Omron CX-Programmer project Китайский_паллетайзер_с_комментариями (CX-Programmer 9.41)

# PLC НовыйПЛК1: CP1E N60

## Global symbols (name address type ; comment)
0.00 BOOL  ; Переключатель Р-А Магазин поддонов
0.01 BOOL  ; КН Магазин поддонов ВНИЗ
0.02 BOOL  ; Маг ВВЕРХ
0.03 BOOL  ; Лапы ОТКР

## Program РВіМРт1 (cyclic task 0)

### Section Сегмент1

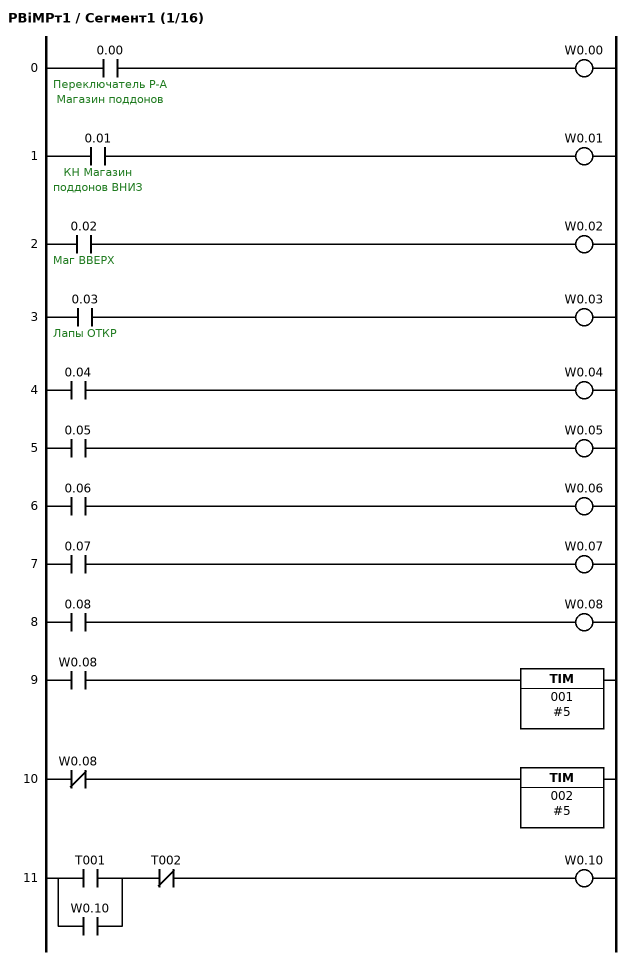
; rung 0
LD 0.00  ; Переключатель Р-А Магазин поддонов
OUT W0.00
; rung 1
LD 0.01  ; КН Магазин поддонов ВНИЗ
OUT W0.01
; rung 2
LD 0.02  ; Маг ВВЕРХ
OUT W0.02
; rung 3
LD 0.03  ; Лапы ОТКР
OUT W0.03
; rung 4
LD 0.04
OUT W0.04
; rung 5
LD 0.05
OUT W0.05
; rung 6
LD 0.06
OUT W0.06
; rung 7
LD 0.07
OUT W0.07
; rung 8
LD 0.08
OUT W0.08
; rung 9
LD W0.08
TIM 001 #5
; rung 10
LDNOT W0.08
TIM 002 #5
; rung 11
LD T001
OR W0.10
ANDNOT T002
OUT W0.10

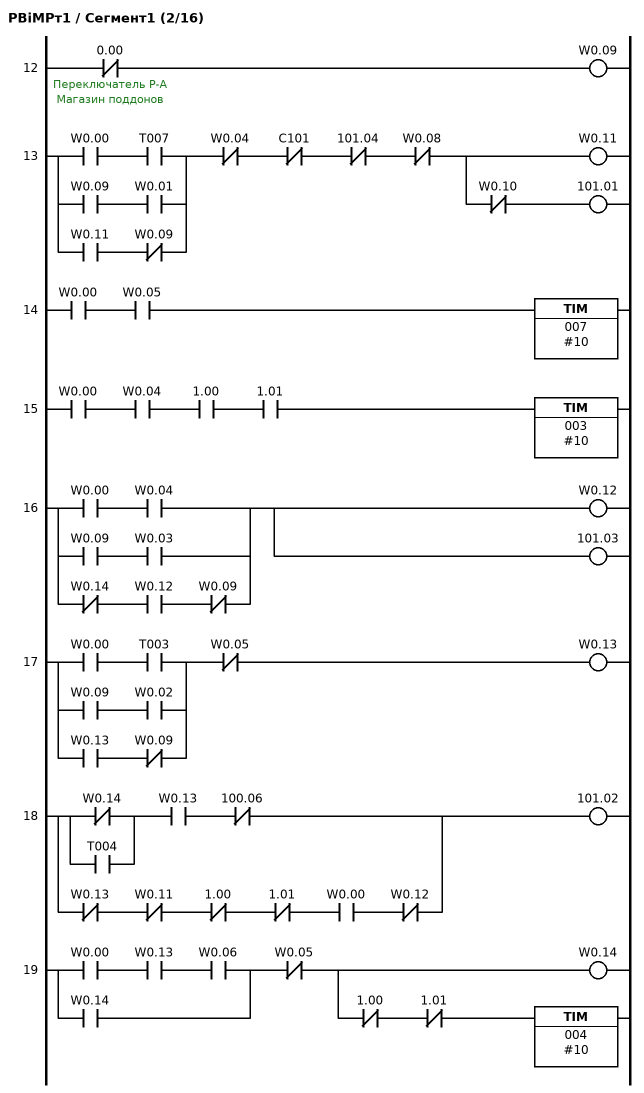
; rung 12
LDNOT 0.00  ; Переключатель Р-А Магазин поддонов
OUT W0.09
; rung 13
LD W0.00
AND T007
LD W0.09
AND W0.01
ORLD
LD W0.11
ANDNOT W0.09
ORLD
ANDNOT W0.04
ANDNOT C101
ANDNOT 101.04
ANDNOT W0.08
OUT W0.11
ANDNOT W0.10
OUT 101.01
; rung 14
LD W0.00
AND W0.05
TIM 007 #10
; rung 15
LD W0.00
AND W0.04
AND 1.00
AND 1.01
TIM 003 #10
; rung 16
LD W0.00
AND W0.04
LD W0.09
AND W0.03
ORLD
LDNOT W0.14
AND W0.12
ANDNOT W0.09
ORLD
OUT W0.12
OUT 101.03
; rung 17
LD W0.00
AND T003
LD W0.09
AND W0.02
ORLD
LD W0.13
ANDNOT W0.09
ORLD
ANDNOT W0.05
OUT W0.13
; rung 18
LDNOT W0.14
OR T004
AND W0.13
ANDNOT 100.06
LDNOT W0.13
ANDNOT W0.11
ANDNOT 1.00
ANDNOT 1.01
AND W0.00
ANDNOT W0.12
ORLD
OUT 101.02
; rung 19
LD W0.00
AND W0.13
AND W0.06
OR W0.14
ANDNOT W0.05
OUT W0.14
ANDNOT 1.00
ANDNOT 1.01
TIM 004 #10

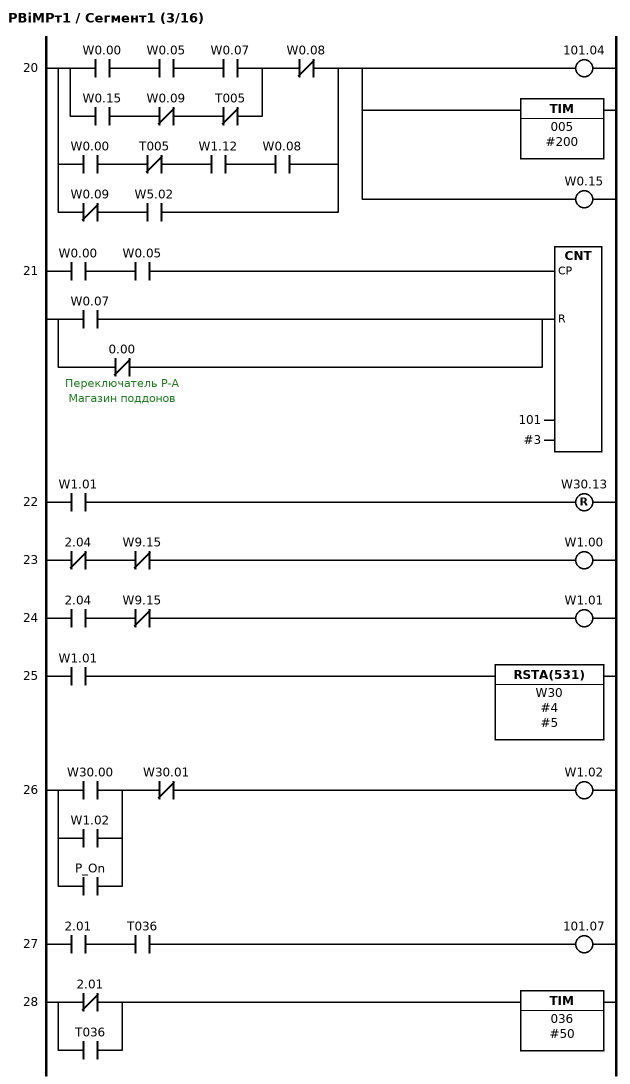
; rung 20
LD W0.00
AND W0.05
AND W0.07
LD W0.15
ANDNOT W0.09
ANDNOT T005
ORLD
ANDNOT W0.08
LD W0.00
ANDNOT T005
AND W1.12
AND W0.08
ORLD
LDNOT W0.09
AND W5.02
ORLD
OUT 101.04
TIM 005 #200
OUT W0.15
; rung 21
LD W0.00
AND W0.05
LD W0.07
ORNOT 0.00  ; Переключатель Р-А Магазин поддонов
CNT 101 #3
; rung 22
LD W1.01
RSET W30.13
; rung 23
LDNOT 2.04
ANDNOT W9.15
OUT W1.00
; rung 24
LD 2.04
ANDNOT W9.15
OUT W1.01
; rung 25
LD W1.01
RSTA(531) W30 #4 #5
; rung 26
LD W30.00
OR W1.02
OR P_On
ANDNOT W30.01
OUT W1.02
; rung 27
LD 2.01
AND T036
OUT 101.07
; rung 28
LDNOT 2.01
OR T036
TIM 036 #50

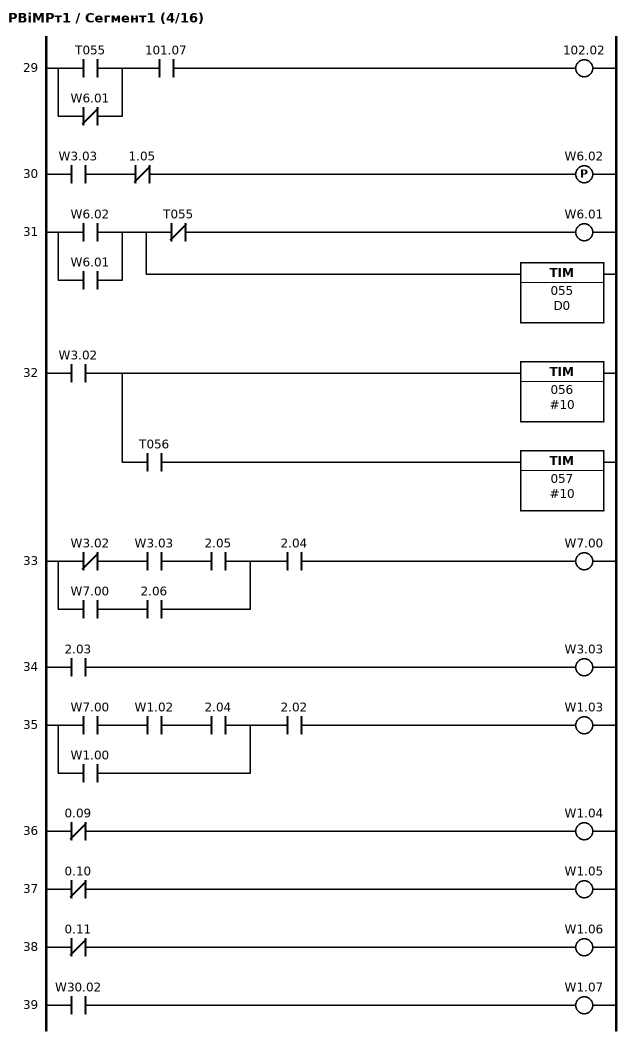
; rung 29
LD T055
ORNOT W6.01
AND 101.07
OUT 102.02
; rung 30
LD W3.03
ANDNOT 1.05
DIFU(013) W6.02
; rung 31
LD W6.02
OR W6.01
OUT TR0
ANDNOT T055
OUT W6.01
LD TR0
TIM 055 D0
; rung 32
LD W3.02
TIM 056 #10
AND T056
TIM 057 #10
; rung 33
LDNOT W3.02
AND W3.03
AND 2.05
LD W7.00
AND 2.06
ORLD
AND 2.04
OUT W7.00
; rung 34
LD 2.03
OUT W3.03
; rung 35
LD W7.00
AND W1.02
AND 2.04
OR W1.00
AND 2.02
OUT W1.03
; rung 36
LDNOT 0.09
OUT W1.04
; rung 37
LDNOT 0.10
OUT W1.05
; rung 38
LDNOT 0.11
OUT W1.06
; rung 39
LD W30.02
OUT W1.07

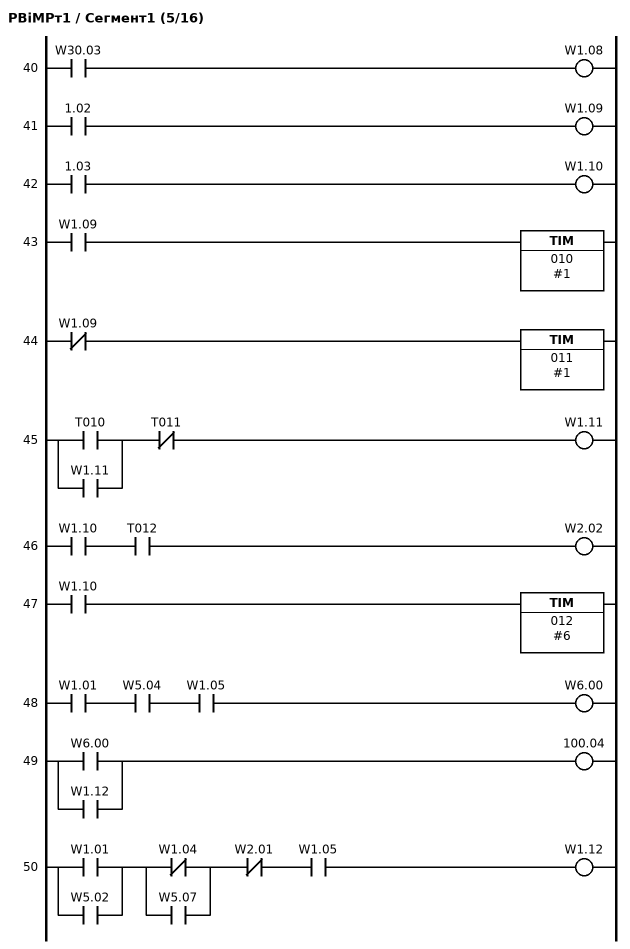
; rung 40
LD W30.03
OUT W1.08
; rung 41
LD 1.02
OUT W1.09
; rung 42
LD 1.03
OUT W1.10
; rung 43
LD W1.09
TIM 010 #1
; rung 44
LDNOT W1.09
TIM 011 #1
; rung 45
LD T010
OR W1.11
ANDNOT T011
OUT W1.11
; rung 46
LD W1.10
AND T012
OUT W2.02
; rung 47
LD W1.10
TIM 012 #6
; rung 48
LD W1.01
AND W5.04
AND W1.05
OUT W6.00
; rung 49
LD W6.00
OR W1.12
OUT 100.04
; rung 50
LD W1.01
OR W5.02
LDNOT W1.04
OR W5.07
ANDLD
ANDNOT W2.01
AND W1.05
OUT W1.12

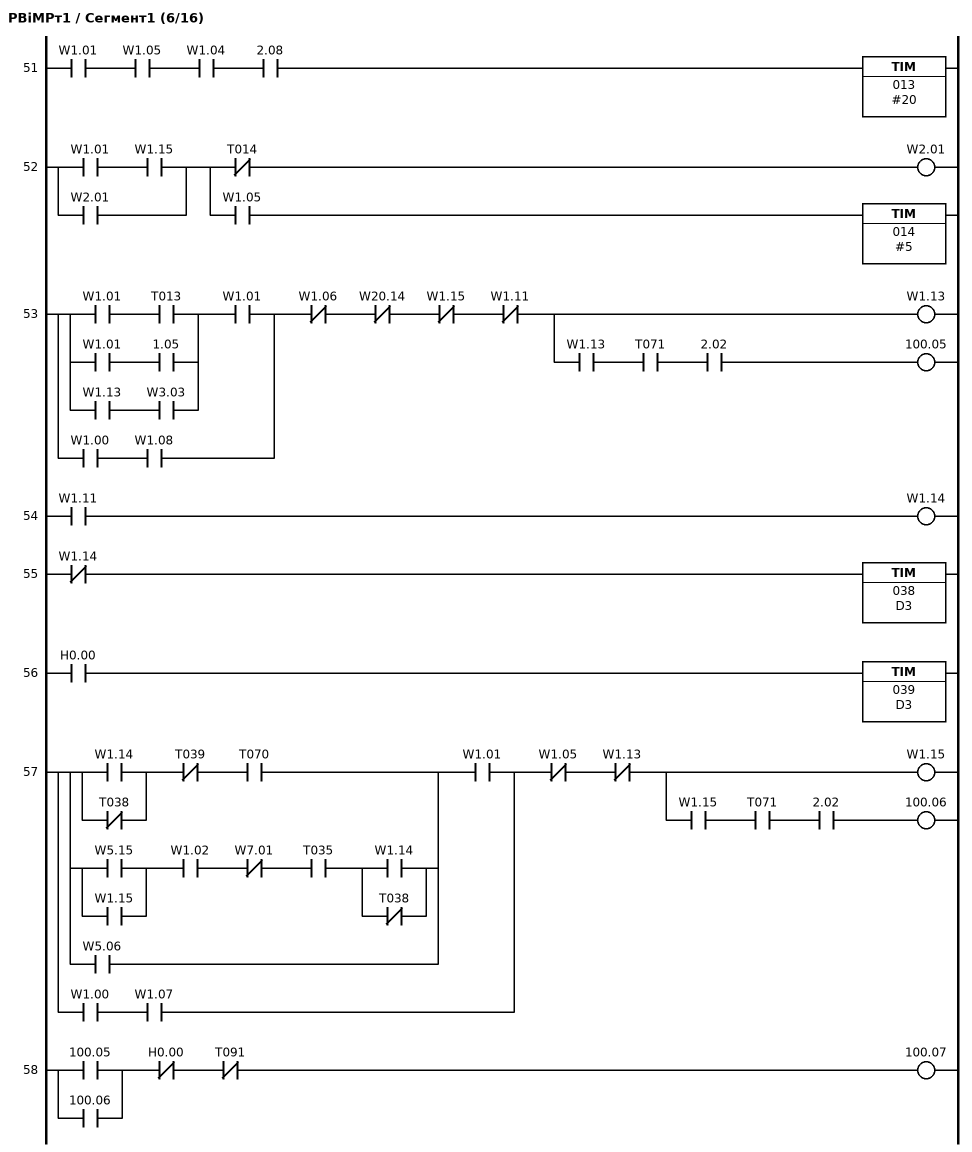
; rung 51
LD W1.01
AND W1.05
AND W1.04
AND 2.08
TIM 013 #20
; rung 52
LD W1.01
AND W1.15
OR W2.01
OUT TR0
ANDNOT T014
OUT W2.01
LD TR0
AND W1.05
TIM 014 #5
; rung 53
LD W1.01
AND T013
LD W1.01
AND 1.05
ORLD
LD W1.13
AND W3.03
ORLD
AND W1.01
LD W1.00
AND W1.08
ORLD
ANDNOT W1.06
ANDNOT W20.14
ANDNOT W1.15
ANDNOT W1.11
OUT W1.13
AND W1.13
AND T071
AND 2.02
OUT 100.05
; rung 54
LD W1.11
OUT W1.14
; rung 55
LDNOT W1.14
TIM 038 D3
; rung 56
LD H0.00
TIM 039 D3
; rung 57
LD W1.14
ORNOT T038
ANDNOT T039
AND T070
LD W5.15
OR W1.15
AND W1.02
ANDNOT W7.01
AND T035
LD W1.14
ORNOT T038
ANDLD
ORLD
OR W5.06
AND W1.01
LD W1.00
AND W1.07
ORLD
ANDNOT W1.05
ANDNOT W1.13
OUT W1.15
AND W1.15
AND T071
AND 2.02
OUT 100.06
; rung 58
LD 100.05
OR 100.06
ANDNOT H0.00
ANDNOT T091
OUT 100.07

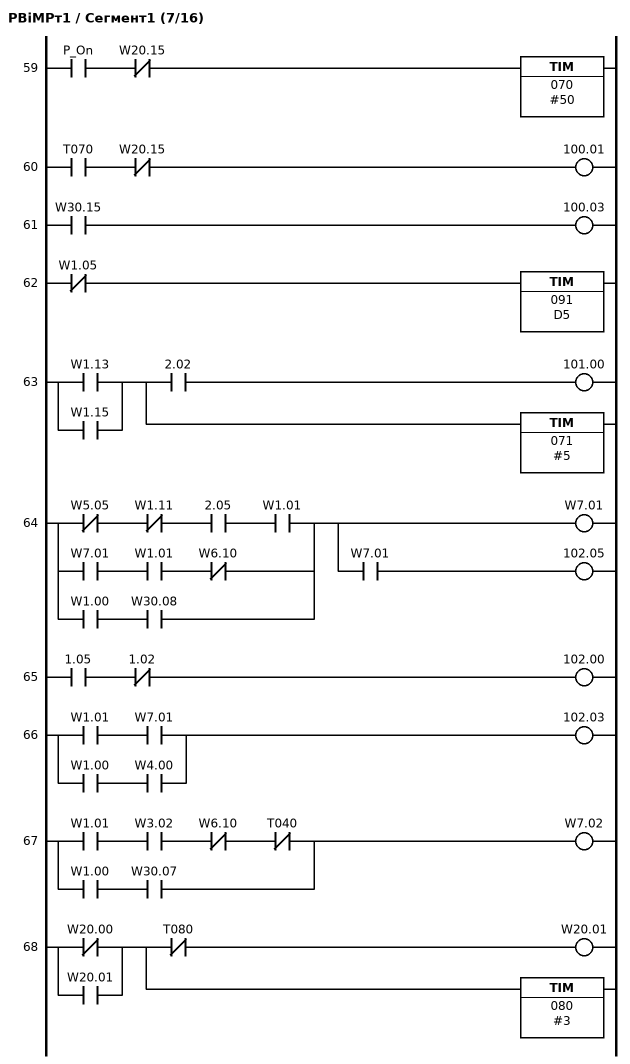
; rung 59
LD P_On
ANDNOT W20.15
TIM 070 #50
; rung 60
LD T070
ANDNOT W20.15
OUT 100.01
; rung 61
LD W30.15
OUT 100.03
; rung 62
LDNOT W1.05
TIM 091 D5
; rung 63
LD W1.13
OR W1.15
OUT TR0
AND 2.02
OUT 101.00
LD TR0
TIM 071 #5
; rung 64
LDNOT W5.05
ANDNOT W1.11
AND 2.05
AND W1.01
LD W7.01
AND W1.01
ANDNOT W6.10
ORLD
LD W1.00
AND W30.08
ORLD
OUT W7.01
AND W7.01
OUT 102.05
; rung 65
LD 1.05
ANDNOT 1.02
OUT 102.00
; rung 66
LD W1.01
AND W7.01
LD W1.00
AND W4.00
ORLD
OUT 102.03
; rung 67
LD W1.01
AND W3.02
ANDNOT W6.10
ANDNOT T040
LD W1.00
AND W30.07
ORLD
OUT W7.02
; rung 68
LDNOT W20.00
OR W20.01
OUT TR0
ANDNOT T080
OUT W20.01
LD TR0
TIM 080 #3

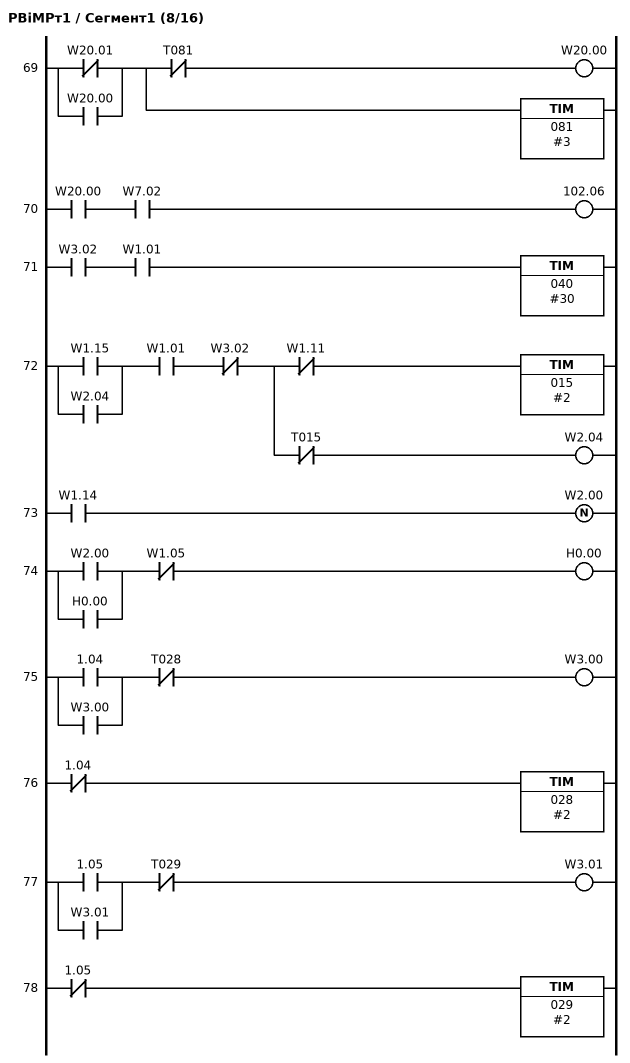
; rung 69
LDNOT W20.01
OR W20.00
OUT TR0
ANDNOT T081
OUT W20.00
LD TR0
TIM 081 #3
; rung 70
LD W20.00
AND W7.02
OUT 102.06
; rung 71
LD W3.02
AND W1.01
TIM 040 #30
; rung 72
LD W1.15
OR W2.04
AND W1.01
ANDNOT W3.02
OUT TR0
ANDNOT W1.11
TIM 015 #2
LD TR0
ANDNOT T015
OUT W2.04
; rung 73
LD W1.14
DIFD(014) W2.00
; rung 74
LD W2.00
OR H0.00
ANDNOT W1.05
OUT H0.00
; rung 75
LD 1.04
OR W3.00
ANDNOT T028
OUT W3.00
; rung 76
LDNOT 1.04
TIM 028 #2
; rung 77
LD 1.05
OR W3.01
ANDNOT T029
OUT W3.01
; rung 78
LDNOT 1.05
TIM 029 #2

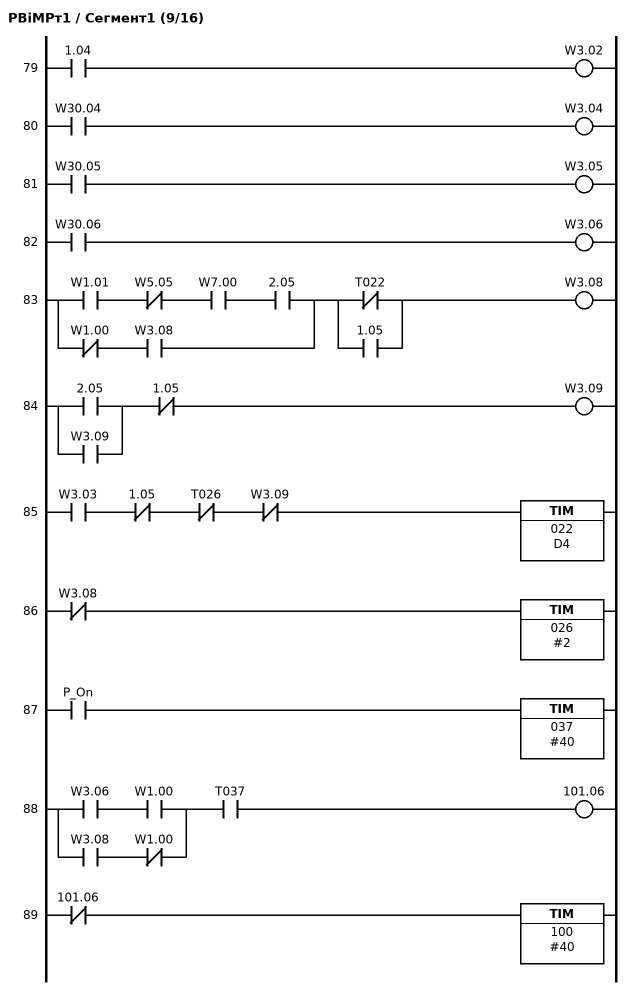
; rung 79
LD 1.04
OUT W3.02
; rung 80
LD W30.04
OUT W3.04
; rung 81
LD W30.05
OUT W3.05
; rung 82
LD W30.06
OUT W3.06
; rung 83
LD W1.01
ANDNOT W5.05
AND W7.00
AND 2.05
LDNOT W1.00
AND W3.08
ORLD
LDNOT T022
OR 1.05
ANDLD
OUT W3.08
; rung 84
LD 2.05
OR W3.09
ANDNOT 1.05
OUT W3.09
; rung 85
LD W3.03
ANDNOT 1.05
ANDNOT T026
ANDNOT W3.09
TIM 022 D4
; rung 86
LDNOT W3.08
TIM 026 #2
; rung 87
LD P_On
TIM 037 #40
; rung 88
LD W3.06
AND W1.00
LD W3.08
ANDNOT W1.00
ORLD
AND T037
OUT 101.06
; rung 89
LDNOT 101.06
TIM 100 #40

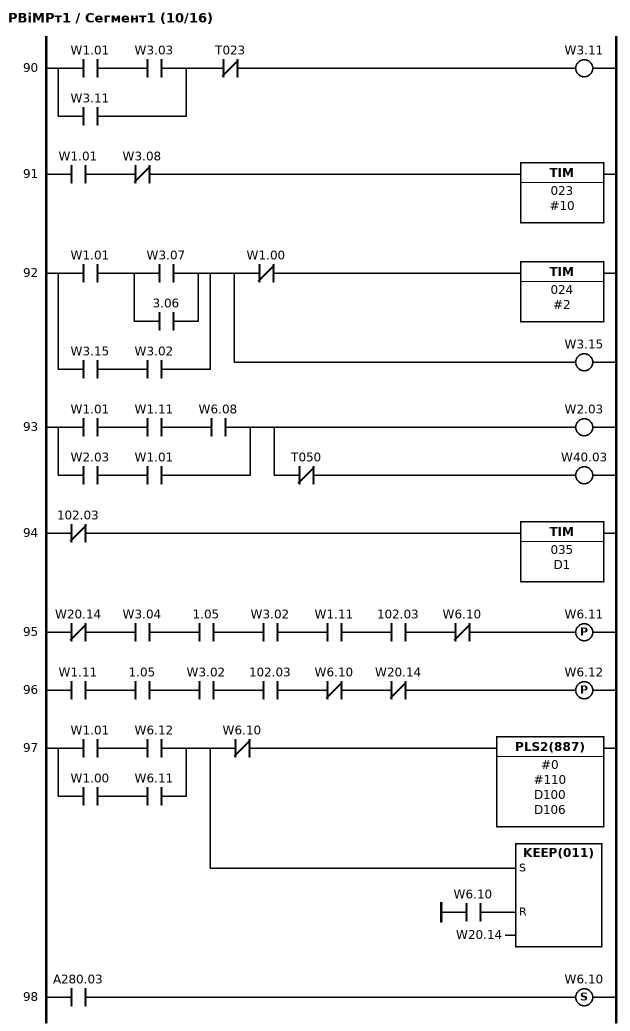
; rung 90
LD W1.01
AND W3.03
OR W3.11
ANDNOT T023
OUT W3.11
; rung 91
LD W1.01
ANDNOT W3.08
TIM 023 #10
; rung 92
LD W1.01
LD W3.07
OR 3.06
ANDLD
LD W3.15
AND W3.02
ORLD
OUT TR0
ANDNOT W1.00
TIM 024 #2
LD TR0
OUT W3.15
; rung 93
LD W1.01
AND W1.11
AND W6.08
LD W2.03
AND W1.01
ORLD
OUT W2.03
ANDNOT T050
OUT W40.03
; rung 94
LDNOT 102.03
TIM 035 D1
; rung 95
LDNOT W20.14
AND W3.04
AND 1.05
AND W3.02
AND W1.11
AND 102.03
ANDNOT W6.10
DIFU(013) W6.11
; rung 96
LD W1.11
AND 1.05
AND W3.02
AND 102.03
ANDNOT W6.10
ANDNOT W20.14
DIFU(013) W6.12
; rung 97
LD W1.01
AND W6.12
LD W1.00
AND W6.11
ORLD
OUT TR0
ANDNOT W6.10
PLS2(887) #0 #110 D100 D106
LD TR0
LD W6.10
KEEP(011) W20.14
; rung 98
LD A280.03
SET W6.10

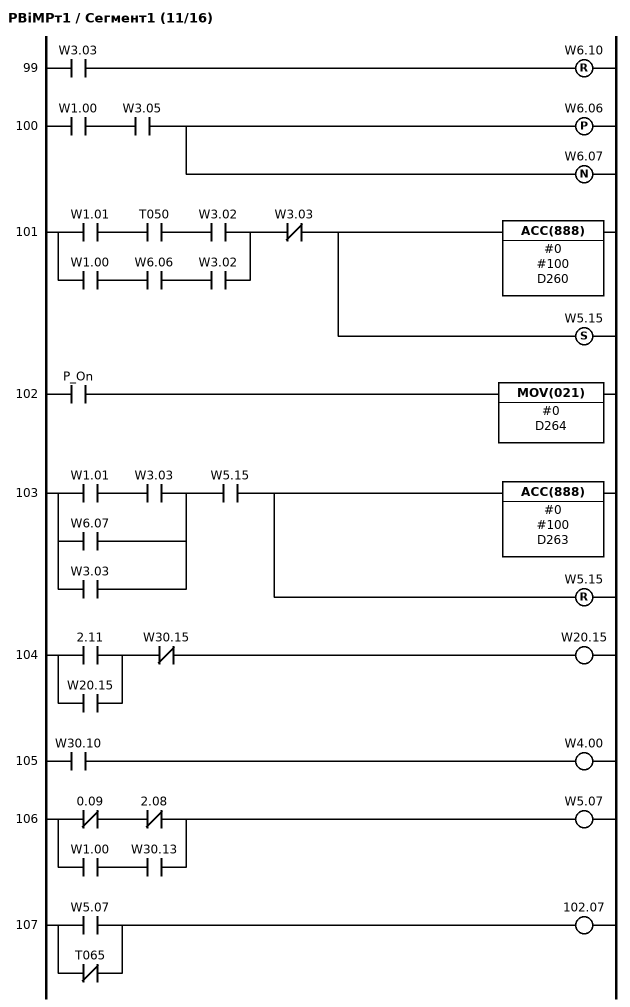
; rung 99
LD W3.03
RSET W6.10
; rung 100
LD W1.00
AND W3.05
DIFU(013) W6.06
DIFD(014) W6.07
; rung 101
LD W1.01
AND T050
AND W3.02
LD W1.00
AND W6.06
AND W3.02
ORLD
ANDNOT W3.03
ACC(888) #0 #100 D260
SET W5.15
; rung 102
LD P_On
MOV(021) #0 D264
; rung 103
LD W1.01
AND W3.03
OR W6.07
OR W3.03
AND W5.15
ACC(888) #0 #100 D263
RSET W5.15
; rung 104
LD 2.11
OR W20.15
ANDNOT W30.15
OUT W20.15
; rung 105
LD W30.10
OUT W4.00
; rung 106
LDNOT 0.09
ANDNOT 2.08
LD W1.00
AND W30.13
ORLD
OUT W5.07
; rung 107
LD W5.07
ORNOT T065
OUT 102.07

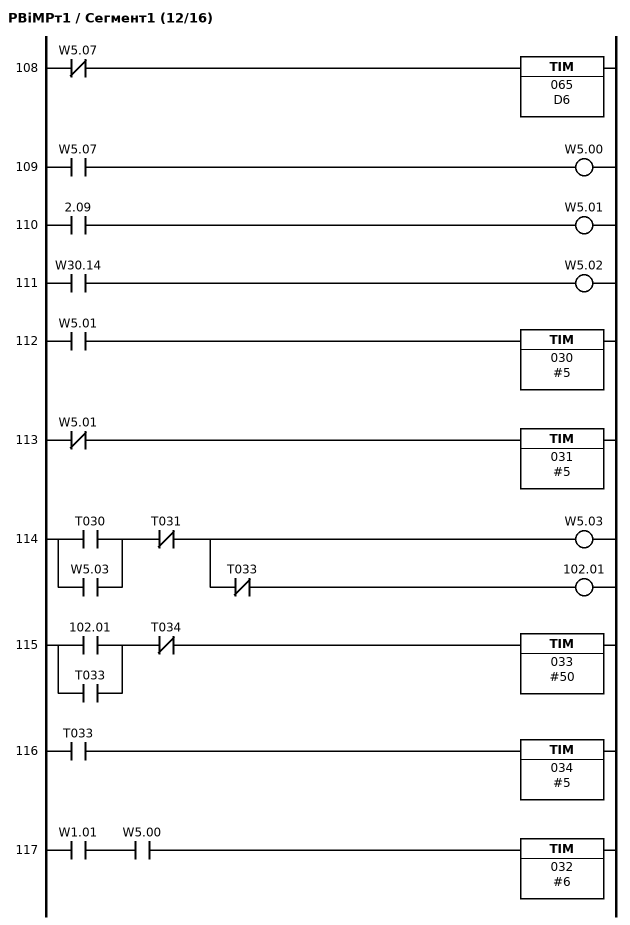
; rung 108
LDNOT W5.07
TIM 065 D6
; rung 109
LD W5.07
OUT W5.00
; rung 110
LD 2.09
OUT W5.01
; rung 111
LD W30.14
OUT W5.02
; rung 112
LD W5.01
TIM 030 #5
; rung 113
LDNOT W5.01
TIM 031 #5
; rung 114
LD T030
OR W5.03
ANDNOT T031
OUT W5.03
ANDNOT T033
OUT 102.01
; rung 115
LD 102.01
OR T033
ANDNOT T034
TIM 033 #50
; rung 116
LD T033
TIM 034 #5
; rung 117
LD W1.01
AND W5.00
TIM 032 #6

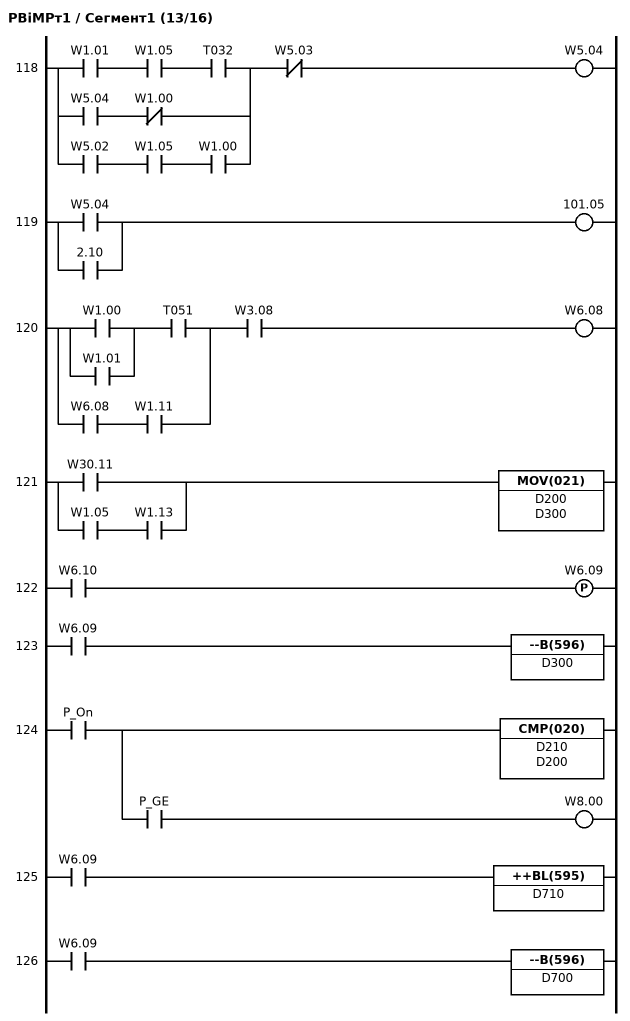
; rung 118
LD W1.01
AND W1.05
AND T032
LD W5.04
ANDNOT W1.00
ORLD
LD W5.02
AND W1.05
AND W1.00
ORLD
ANDNOT W5.03
OUT W5.04
; rung 119
LD W5.04
OR 2.10
OUT 101.05
; rung 120
LD W1.00
OR W1.01
AND T051
LD W6.08
AND W1.11
ORLD
AND W3.08
OUT W6.08
; rung 121
LD W30.11
LD W1.05
AND W1.13
ORLD
MOV(021) D200 D300
; rung 122
LD W6.10
DIFU(013) W6.09
; rung 123
LD W6.09
--B(596) D300
; rung 124
LD P_On
CMP(020) D210 D200
AND P_GE
OUT W8.00
; rung 125
LD W6.09
++BL(595) D710
; rung 126
LD W6.09
--B(596) D700

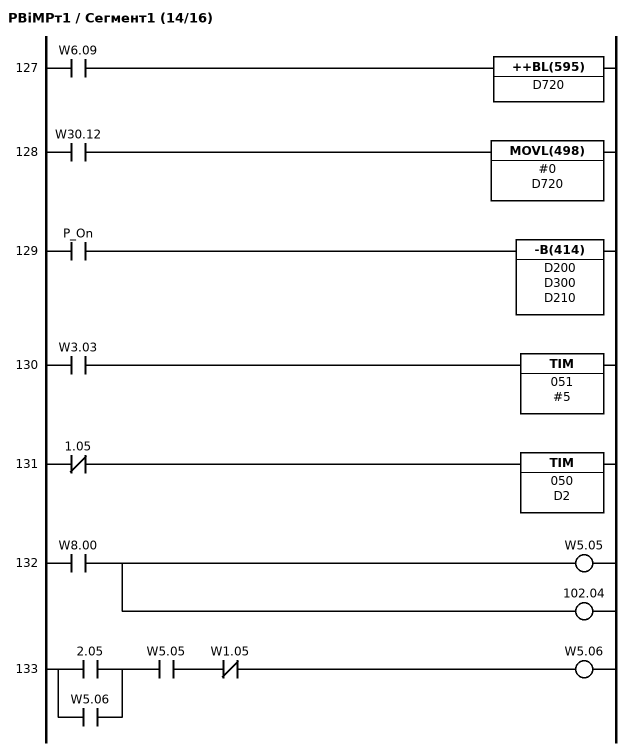
; rung 127
LD W6.09
++BL(595) D720
; rung 128
LD W30.12
MOVL(498) #0 D720
; rung 129
LD P_On
-B(414) D200 D300 D210
; rung 130
LD W3.03
TIM 051 #5
; rung 131
LDNOT 1.05
TIM 050 D2
; rung 132
LD W8.00
OUT W5.05
OUT 102.04
; rung 133
LD 2.05
OR W5.06
AND W5.05
ANDNOT W1.05
OUT W5.06

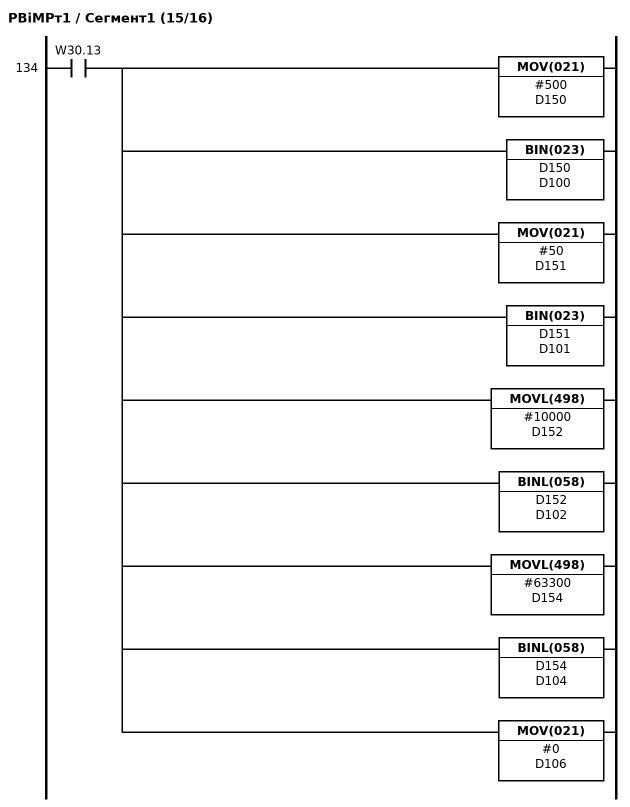
; rung 134
LD W30.13
MOV(021) #500 D150
BIN(023) D150 D100
MOV(021) #50 D151
BIN(023) D151 D101
MOVL(498) #10000 D152
BINL(058) D152 D102
MOVL(498) #63300 D154
BINL(058) D154 D104
MOV(021) #0 D106

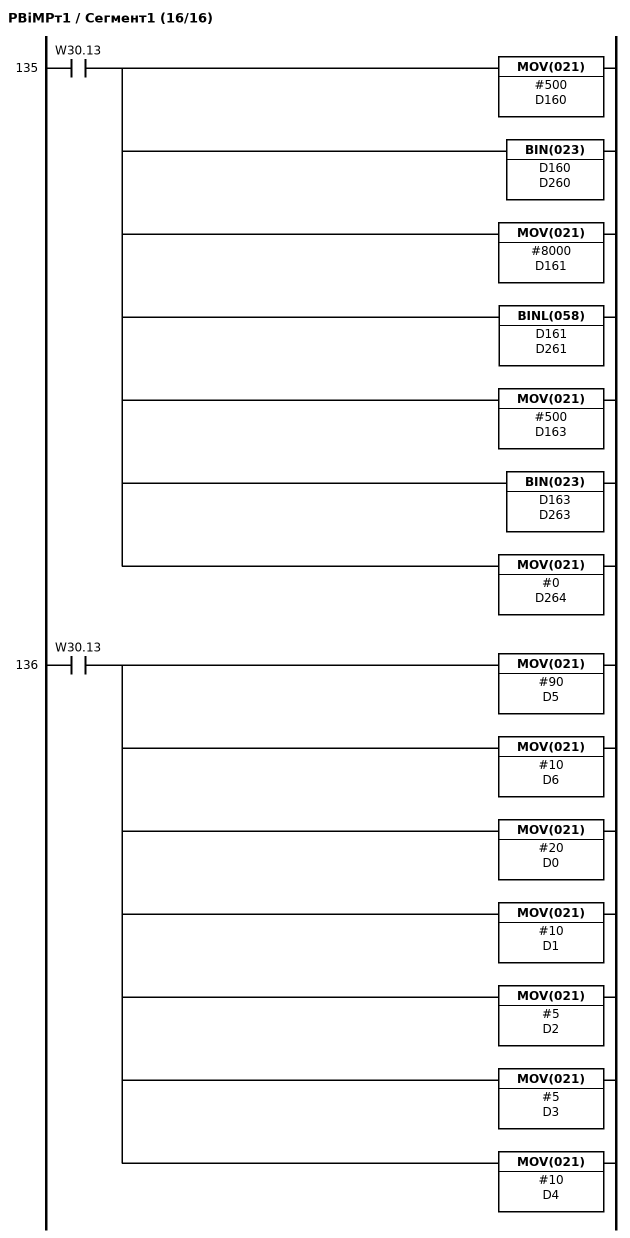
; rung 135
LD W30.13
MOV(021) #500 D160
BIN(023) D160 D260
MOV(021) #8000 D161
BINL(058) D161 D261
MOV(021) #500 D163
BIN(023) D163 D263
MOV(021) #0 D264
; rung 136
LD W30.13
MOV(021) #90 D5
MOV(021) #10 D6
MOV(021) #20 D0
MOV(021) #10 D1
MOV(021) #5 D2
MOV(021) #5 D3
MOV(021) #10 D4
; rung 137
END(001)